TYPE HMIInterfaceOperatingMode :
STRUCT
	PLCToHMI	:	PLCToHMIOperatingMode;
	HMIToPLC	:	HMIToPLCOperatingMode;
END_STRUCT
END_TYPE

(* stored: Version 1.1.0.1
   DUT HMIInterfaceOperatingMode: Id {79f78aa5-5406-4384-8bf8-b6e18272cd9d} *)
